// TIA Portal V19 export
DATA_BLOCK "LB113"   // DB80
// stored: InstanceOfName ButtonsSafe_LB113, InstanceOfType FB
"ButtonsSafe_LB113"
   // VAR_INPUT
   //    Reset_OthersPBs_Activation_IN : Bool;
   // END_VAR
   // VAR_OUTPUT
   //    Reset_OthersPBs_Activation_OUT : Bool;
   // END_VAR
   // VAR
   //    i : Int;
   //    iOperation : Int;
   //    iConcurrentOperation : Int;
   //    SettingWriteDone : Bool;
   //    PbPanel : "Buttons2Hands";
   //    PB : Struct
   //       ResetAlarms : Bool;
   //       JBPinchroll_Fwd : Bool;
   //       JBPinchroll_Bwd : Bool;
   //       JBCutCycle : Bool;
   //       Straightener_Fwd : Bool;
   //       Straightener_Bwd : Bool;
   //    END_STRUCT;
   // END_VAR
BEGIN
END_DATA_BLOCK
